TYPE
    TcoSmartFunctionKitConfig :
    STRUCT
        DataFormat : eTcoDataFormat := TcoUtilities.eTcoDataFormat.BigEndian;
        InfoTime : TIME := T#2S;
        ErrorTime : TIME := T#5S;
    END_STRUCT
END_TYPE

(* stored: Version 1.1.0.1
   DUT TcoSmartFunctionKitConfig: Id {e14a5d54-2aa1-4e00-8fb0-64bc9475e2ad} *)
